FUNCTION_BLOCK FB_RetainedData
VAR_INPUT
	xSaveAll								: BOOL;
END_VAR
VAR_OUTPUT
	xReadComplete							: BOOL;
	xErr									: BOOL;
	nErrID									: UDINT;
	RecipeSaveDone: BOOL;
END_VAR
VAR
	//fbRetainGlobalSettings					: FB_Retain;
	fbRetainRecipes							: FB_Retain;
	
	xAllRead								: BOOL;
	tonFileReadComplete						: ton;
	testbit: BOOL;
END_VAR

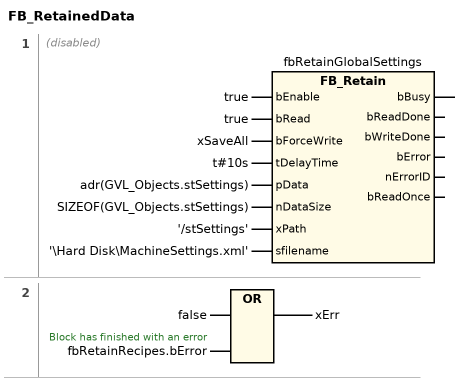
// NETWORK 1 (disabled)
// fbRetainGlobalSettings(
//     bEnable := true,
//     bRead := true,
//     bForceWrite := xSaveAll,
//     tDelayTime := t#10s,
//     pData := adr(GVL_Objects.stSettings),
//     nDataSize := SIZEOF(GVL_Objects.stSettings),
//     xPath := '/stSettings',
//     sfilename := '\Hard Disk\MachineSettings.xml'); // FB_Retain

// NETWORK 2
//   fbRetainRecipes.bError: Block has finished with an error
xErr := false OR fbRetainRecipes.bError;

END_FUNCTION_BLOCK

(* stored: Version 1.1.0.1, ProductVersion 3.1.4020.12
   POU FB_RetainedData: Id {70bd72c8-8d24-4e06-948e-b7c23ef50e23}, SpecialFunc None *)
